FUNCTION_BLOCK FB_PhotonEnergy
VAR_INPUT
    Undulator : I_UndulatorComplex;
END_VAR
VAR_OUTPUT
END_VAR
VAR_IN_OUT
    BP : ST_BeamParams;
END_VAR
VAR
    nCurrentPhotonEnergyBitmask : UDINT;
    nTargetPhotonEnergyBitmask : UDINT;
END_VAR


//Update BP
nCurrentPhotonEnergyBitmask := F_eVRangeCalculator(Undulator.rCurrentPhotonEnergy, nCurrentPhotonEnergyBitmask);
nTargetPhotonEnergyBitmask := F_eVRangeCalculator(Undulator.rTargetPhotonEnergy, nTargetPhotonEnergyBitmask);

BP.neVRange := nCurrentPhotonEnergyBitmask OR nTargetPhotonEnergyBitmask;

END_FUNCTION_BLOCK

(* stored: Version 1.1.0.1
   POU FB_PhotonEnergy: Id {3bff9277-6cb3-4e5b-8a82-abf3351b7c37}, SpecialFunc None *)
